FUNCTION_BLOCK AX_TONOF (* Standard timer function block (on/off-delay timing) *)
  (* Standard: 61499-2; Classification: standard timer function block; Description: Copyright (c) 2024 HR Agrartechnik GmbH This program and the accompanying materials are made available under the terms of the Eclipse Public License 2.0 which is available at https://www.eclipse.org/legal/epl-2.0/ SPDX-License-Identifier: EPL-2.0 AX_TONOF -- On/Off-delay timer FB with AX adapter interface The adapter input IN triggers execution (E1->REQ) and provides the boolean input value (D1->IN). The event input R presets both delay times PT_ON and PT_OFF and resets the timer. When IN goes TRUE, Q becomes TRUE after delay PT_ON. When IN goes FALSE, Q becomes FALSE after delay PT_OFF. Reset stops both timers and sets Q to FALSE. *)
  (* Version 3.0, 2025-04-14, Patrick Aigner, changed package *)
  (* Version 1.1, 2024-04-23, Franz Höpfinger, HR Agrartechnik GmbH, Add a Reset to Timer FBs *)
  (* Version 1.0, 2024-03-04, Franz Höpfinger, HR Agrartechnik GmbH *)
  PACKAGE adapter::events::unidirectional::timers;
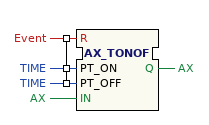
  EVENT_INPUT
    R WITH PT_ON, PT_OFF; (* Reset *)
  END_EVENT
  VAR_INPUT
    PT_ON : TIME; (* ON delay time *)
    PT_OFF : TIME; (* OFF delay time *)
  END_VAR
  SOCKETS
    IN : adapter::types::unidirectional::AX; (* Timer input (AX adapter) *)
  END_SOCKETS
  PLUGS
    Q : adapter::types::unidirectional::AX; (* Timer output (AX adapter) *)
  END_PLUGS
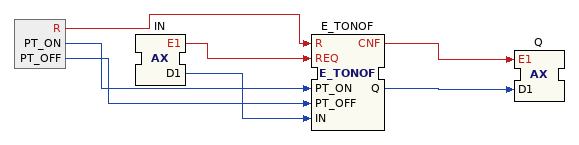
  FBS
    E_TONOF : iec61499::events::timers::E_TONOF;
  END_FBS
  EVENT_CONNECTIONS
    R TO E_TONOF.R;
    IN.E1 TO E_TONOF.REQ;
    E_TONOF.CNF TO Q.E1;
  END_CONNECTIONS
  DATA_CONNECTIONS
    PT_ON TO E_TONOF.PT_ON;
    PT_OFF TO E_TONOF.PT_OFF;
    IN.D1 TO E_TONOF.IN;
    E_TONOF.Q TO Q.D1;
  END_CONNECTIONS
END_FUNCTION_BLOCK
